(* PLC project  *)

CONFIGURATION FSOE_3
END_CONFIGURATION
